Staubli VAL3: Recorder.dtx

mdesc mNomSpeed
num nFileHandle
string sFile
public bool bRecord
